{attribute 'GeneratedUsingTerminal: EL6601--0000'}
{attribute addProperty BoxType "EL6601--0000"}
{attribute addProperty Id "InfoDataAT %I*InfoData_94A18F5E2"}
{attribute addProperty CRC "2009557638"}
{attribute addProperty Size "2"}
TYPE EL6601_77C76A86 EXTENDS EtcSlaveTerminalBase_947E5A46 :
STRUCT
	{attribute addProperty Name "InfoData"}
	InfoData : InfoData_94A18F5E;
END_STRUCT
END_TYPE

(* stored: Version 1.2.0.0, ProductVersion 3.1.4024.9
   DUT EL6601_77C76A86: Id {bc24b534-4228-42e9-af8e-c1694fd0343a} *)
